// TIA Portal project "CONTADOR HORAS TOTAL Y PARCIAL" (V11)

(* hardware
DEVICE "S7300/ET200 station_1"  SIMATIC 300-Station
   slot 0: "Perfil soporte_0"  Rail  6ES7 390-1***0-0AA0
   slot 2: "PLC_1"  CPU 313C-2 DP  6ES7 313-6CF03-0AB0  V2.6
      slot 0: "Interfaz MPI_1"  MPI
      slot 1: "Interfaz DP_1"  DP
      slot 2: "DI16/DO16_1"  DI16/DO16
      slot 4: "Contaje_1"  Counter
*)

// ===== PLC "PLC_1"  CPU 313C-2 DP =====

VAR_GLOBAL   // PLC tag table "Tabla de variables estándar"
   "MARCHA" AT %E0.0 : Bool;
   "PARO" AT %I0.1 : Bool;
   "SG.T" AT %MW10 : Int;
   "MIN.T" AT %MW12 : Int;
   "HORAS.T" AT %MD14 : DInt;
   "SG.P" AT %MW20 : Int;
   "MIN.P" AT %MW22 : Int;
   "HORAS.P" AT %MD24 : DInt;
   "Tag_1" AT %MW14 : Int;
END_VAR

DATA_BLOCK "CONTADOR HORAS T Y PARCIAL_DB"   // DB1
{ S7_Optimized_Access := 'FALSE' }
VERSION : 0.1
// stored: InstanceOfName CONTADOR HORAS T Y PARCIAL
"CONTADOR HORAS T Y PARCIAL"
BEGIN
END_DATA_BLOCK

FUNCTION_BLOCK "CONTADOR HORAS T Y PARCIAL"   // FB1, LAD
{ S7_Optimized_Access := 'FALSE' }
VERSION : 0.1
   VAR_INPUT
      MARCHA : Bool;
      PARO : Bool;
      "TIM 1" : Timer;
      "TIM 2" : Timer;
   END_VAR
   VAR_OUTPUT
      "SG.T" : Int;
      "MIN-T" : Int;
      "HORAS.T" : DInt;
      "SG.P" : Int;
      "MIN.P" : Int;
      "HORAS.P" : DInt;
   END_VAR
   VAR
      B0 : Bool;
      B1 : Bool;
      B2 : Bool;
      B3 : Bool;
      B4 : Bool;
      B5 : Bool;
      B6 : Bool;
      B7 : Bool;
      F10 : Bool;
      F11 : Bool;
      F12 : Bool;
      F13 : Bool;
      F14 : Bool;
      F15 : Bool;
      F16 : Bool;
      F17 : Bool;
      F20 : Bool;
      F21 : Bool;
      F22 : Bool;
      F23 : Bool;
      F24 : Bool;
      F25 : Bool;
   END_VAR
BEGIN
END_FUNCTION_BLOCK

ORGANIZATION_BLOCK "Main"   // OB1, LAD
TITLE = "Main Program Sweep (Cycle)"
{ S7_Optimized_Access := 'FALSE' }
VERSION : 0.1
   VAR_TEMP
      OB1_EV_CLASS : Byte;   // Bits 0-3 = 1 (Coming event), Bits 4-7 = 1 (Event class 1)
      OB1_SCAN_1 : Byte;   // 1 (Cold restart scan 1 of OB 1), 3 (Scan 2-n of OB 1)
      OB1_PRIORITY : Byte;   // Priority of OB Execution
      OB1_OB_NUMBR : Byte;   // 1 (Organization block 1, OB1)
      OB1_RESERVED_1 : Byte;   // Reserved for system
      OB1_RESERVED_2 : Byte;   // Reserved for system
      OB1_PREV_CYCLE : Int;   // Cycle time of previous OB1 scan (milliseconds)
      OB1_MIN_CYCLE : Int;   // Minimum cycle time of OB1 (milliseconds)
      OB1_MAX_CYCLE : Int;   // Maximum cycle time of OB1 (milliseconds)
      OB1_DATE_TIME : Date_And_Time;   // Date and time OB1 started
   END_VAR
BEGIN

REGION Network 1
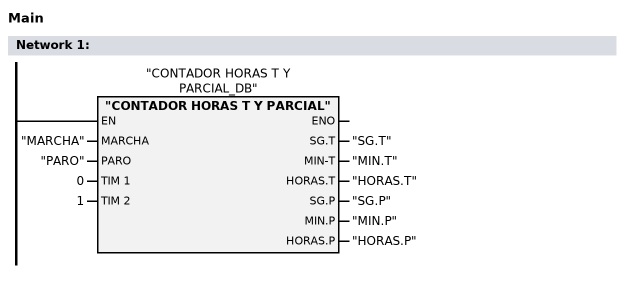
   RUNG wire#powerrail
      "CONTADOR HORAS T Y PARCIAL_DB"(MARCHA := "MARCHA", PARO := "PARO", "TIM 1" := 0, "TIM 2" := 1, "SG.T" => "SG.T", "MIN-T" => "MIN.T", "HORAS.T" => "HORAS.T", "SG.P" => "SG.P", "MIN.P" => "MIN.P", "HORAS.P" => "HORAS.P")
   END_RUNG
   // the same network as SCL:
   "CONTADOR HORAS T Y PARCIAL_DB"(MARCHA := "MARCHA",   // "CONTADOR HORAS T Y PARCIAL"
                           PARO := "PARO",
                           "TIM 1" := 0,
                           "TIM 2" := 1,
                           "SG.T" => "SG.T",
                           "MIN-T" => "MIN.T",
                           "HORAS.T" => "HORAS.T",
                           "SG.P" => "SG.P",
                           "MIN.P" => "MIN.P",
                           "HORAS.P" => "HORAS.P");
END_REGION
END_ORGANIZATION_BLOCK